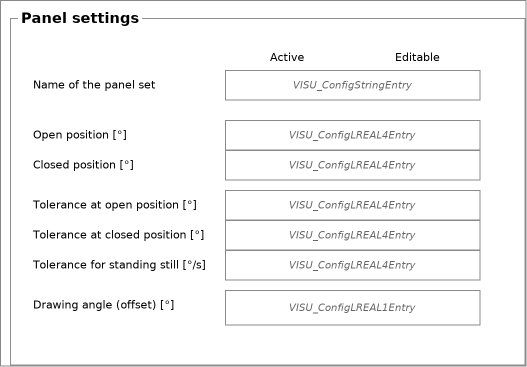
VISUALIZATION VISU_CoverConfig_Panel  // 527x367
VAR_IN_OUT
	activeConfig : CoverPanelConfig;
	editableConfig : CoverPanelConfig;
END_VAR
    GroupBox (10,10 515x355), "Panel settings"
        Label (345,35 125x25), "Editable"
        Label (215,35 125x25), "Active"
        Frame (215,60 255x30)
            shows VISU_ConfigStringEntry(active := activeConfig.name, editable := editableConfig.name)
        Label (20,60 175x30), "Name of the panel set"
        Label (20,210 190x30), "Tolerance at closed position [°]"
        Label (20,240 175x30), "Tolerance for standing still [°/s]"
        Label (20,180 175x30), "Tolerance at open position [°]"
        Label (20,140 175x30), "Closed position [°]"
        Label (20,110 175x30), "Open position [°]"
        Frame (215,110 255x30)
            shows VISU_ConfigLREAL4Entry(active := activeConfig.openPosition, editable := editableConfig.openPosition)
        Frame (215,140 255x30)
            shows VISU_ConfigLREAL4Entry(active := activeConfig.closedPosition, editable := editableConfig.closedPosition)
        Frame (215,180 255x30)
            shows VISU_ConfigLREAL4Entry(active := activeConfig.openTolerance, editable := editableConfig.openTolerance)
        Frame (215,210 255x30)
            shows VISU_ConfigLREAL4Entry(active := activeConfig.closedTolerance, editable := editableConfig.closedTolerance)
        Frame (215,240 255x30)
            shows VISU_ConfigLREAL4Entry(active := activeConfig.standstillTolerance, editable := editableConfig.standstillTolerance)
        Label (20,280 195x30), "Drawing angle (offset) [°]"
        Frame (215,280 255x35)
            shows VISU_ConfigLREAL1Entry(active := activeConfig.offset, editable := editableConfig.offset)
END_VISUALIZATION

(* stored: Version 1.1.0.1, ProductVersion 3.1.4019.2
   Visu VISU_CoverConfig_Panel: Id {ef51bf21-b27b-43fe-bfd6-60c2a60c49d8} *)
